Omron CX-Programmer project NewProject (CX-Programmer 9.73)

# PLC NewPLC1: CP1E N40

## Global symbols (name address type ; comment)
0.00 BOOL  ; green button
100.05 BOOL  ; green light
1.11 BOOL  ; red butoon

## Program NewProgram1 (cyclic task 0)

### Section Section1

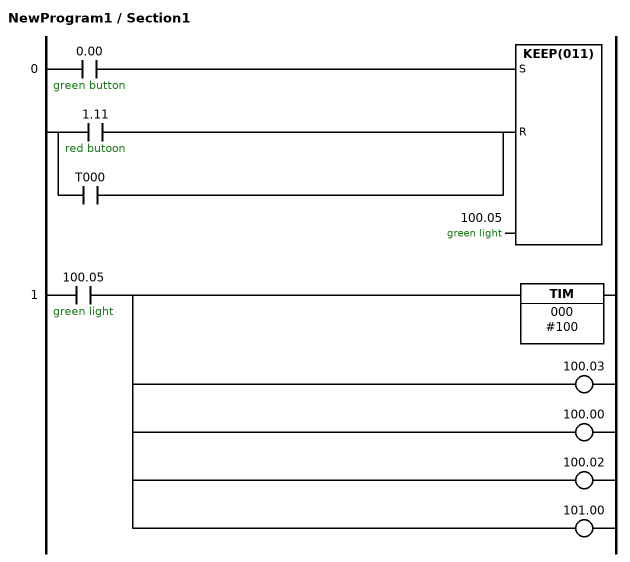
; rung 0
LD 0.00  ; green button
LD 1.11  ; red butoon
OR T000
KEEP(011) 100.05  ; green light
; rung 1
LD 100.05  ; green light
TIM 000 #100
OUT 100.03
OUT 100.00
OUT 100.02
OUT 101.00

### Section END
; rung 0
END(001)